(* Logix 5000 project; controller PBS_Perfusion vendor 1 type 14 code 217 rev 32.14; software revision 32.03; part 18 of 27 *)
(* tags used below, declared in another part *)
   Inp_OpenLS : BOOL;   // Valve Open Limit Switch 1=confirmed fully open
   Inp_ClosedLS : BOOL;   // Valve Closed Limit Switch 1=confirmed fully closed
   Inp_ActuatorFault : BOOL;   // Valve Actuator Fault (overload, etc.), 0=OK, 1=Fault)
   Inp_IntlkOK : BOOL;   // 1=Interlocks OK, Pulse Output Valve can be moved
   Inp_NBIntlkOK : BOOL;   // 1=Non-Bypassable Interlocks OK, Pulse Output Valve can be moved
   Inp_IntlkAvail : BOOL;   // 1 = Interlock Availibility OK
   Inp_IOFault : BOOL;   // Input / Output Communication Status 0=OK, 1=fail
   Inp_Sim : BOOL;   // 1=I/O are being simulated, set output CV to 0.0, ignore I/O Fault
   Inp_Reset : BOOL;   // 1=Reset shed latches and cleared alarms
   Cfg_ShedHold : BOOL;   // 1=Hold Output on Interlock or bad PV, 0=Go to Cfg_IntlkCV
   Cfg_ShedOnIOFault : BOOL;   // 1=Take shed action (hold or interlock CV) on I/O Fault
   Cfg_SkipRoCLim : BOOL;   // 1=Skip RoC Limiting in Intlk, Maint, Ovrd modes
   Cfg_SetTrack : BOOL;   // 1=PSets track OSets in Oper, OSets track PSets in Prog, 0=no tracking
   Cfg_SetTrackOvrdHand : BOOL;   // 1=Prog/Oper Settings track Override/Hand CV
   Cfg_HasOpenLS : BOOL;   // 1=Valve provides an Open Limit Switch signal
   Cfg_HasClosedLS : BOOL;   // 1=Valve provides a Closed Limit Switch signal
   Cfg_UseOpenLS : BOOL;   // 1=Valve Open LS should be used for open/closed status
   Cfg_UseClosedLS : BOOL;   // 1=Valve Closed LS should be used for open/closed status
   Cfg_LSFail : BOOL;   // 1=both switches ON=fail, 0=both switches OFF=fail
   Cfg_MinCV : REAL;   // Minimum CV (in CV EU, for limiting)
   Cfg_MaxCV : REAL;   // Maximum CV (in CV EU, for limiting)
   Cfg_CVRoCLimInc : REAL;   // CV Rate of Change Limit, Increasing, (EU/sec, 0=unlimited)
   Cfg_CVRoCLimDec : REAL;   // CV Rate of Change Limit, Decreasing, (EU/sec, 0=unlimited)
   Cfg_IntlkCV : REAL;   // CV (target in EU) when interlocked (if not Cfg_ShedHold)
   Cfg_CVEUMin : REAL;   // CV Minimum in Engineering Units (for scaling)
   Cfg_CVEUMax : REAL;   // CV Maximum in Engineering Units (for scaling)
   Cfg_CVRawMin : REAL;   // CV Minimum in I/O (raw) Units (for scaling)
   Cfg_CVRawMax : REAL;   // CV Maximum in I/O (raw) Units (for scaling)
   Cfg_CycleT : REAL;   // Open and Close Pulse Output overall period (s)
   Cfg_OpenRate : REAL;   // Rate at which valve moves when opening (CV EU/sec)
   Cfg_CloseRate : REAL;   // Rate at which valve moves when closing (CV EU/sec)
   Cfg_MaxOnT : REAL;   // Open and Close Pulse Output maximum ON time (s)
   Cfg_MinOnT : REAL;   // Open and Close Pulse Output minimum ON time (s)
   Cfg_BumpT : REAL;   // Time to bump valve open or closed (by Oper) when Fdbk Bad (sec)
   Cfg_Deadtime : REAL;   // Additional time on first pulse after stop or direction change
   Cfg_MaxClosedPos : REAL;   // Position above which valve is assumed open if limit switches not used
   PSet_CV : REAL;   // Program Setting of Controlled Variable (output) (CV EU)
   XSet_CV : REAL;   // External Setting of Controlled Variable (output) (CV EU)
   PCmd_Reset : BOOL;   // Program Command to reset shed latches and cleared alarms
   XCmd_Reset : BOOL;   // External Command to reset shed latches and cleared alarms
   Out_CV : REAL;   // CV Output in Raw (I/O Card) Units
   Out_Open : BOOL;   // Pulse Output to drive valve Open
   Out_Close : BOOL;   // Pulse Output to drive valve closed
   Val_Pos : REAL;   // Valve actual position from feedback (CV EU)
   Val_CVSet : REAL;   // Value of selected CV Setting (before rate limiting, CV EU)
   Val_CVOut : REAL;   // Value of CV output (after clamping and ramping) (CV EU)
   SrcQ_IO : DINT;   // Source and Quality of primary I/O (enumeration)
   SrcQ : DINT;   // Source and Quality of primary Val/Sts (enumeration)
   Val_Fdbk : DINT;   // Device Feedback 0=Moving, 1=Closed, 2=Opened, 3=Limit Switch Failure
   Val_Sts : DINT;   // 0=AtTarget, 1=RampClose, 2=RampOpen, 3=Clamp@Min, 4=Clamp@Max, 5=BumpClose, 6=BumpOpen
   Val_Fault : DINT;   // Device Fault Status 0=none, 32=I/OFault, 34=CfgErr
   Val_NotifyAll : DINT;   // Highest Alarm prio and ack status this object + channel (enum)
   Val_UnackAlmC : DINT;   // Count of Unacknowledged Alarms
   Sts_CVInfNaN : BOOL;   // 1=Selected CV is Infinite or Not A Number (1.$, 1.#NaN)
   Sts_PosInfNaN : BOOL;   // 1=Inp_PosFdbk is Infinite or Not A Number (1.$, 1.#NaN)
   Sts_BumpOpen : BOOL;   // 1=Bump Open Requested or Active
   Sts_BumpClose : BOOL;   // 1=Bump Close Requested or Active
   Sts_Ramping : BOOL;   // 1=CV is ramping to target
   Sts_Clamped : BOOL;   // 1=CV Set is clamped at CVMin or CVMax
   Sts_SkipRoCLim : BOOL;   // 1=Rate of Change Limiting was skipped this scan (Maint, Ovrd, Intlk, Hand)
   Sts_Active : BOOL;   // 1=CV is greater than Cfg_MaxClosedPos, show valve symbol as "opened"
   Sts_Available : BOOL;   // 1=Pulse Output Valve available for control by automation (Prog)
   Sts_BypActive : BOOL;   // 1=Bypassing Active (Bypassed or Maintenance)
   Sts_LSFail : BOOL;   // 1=Limit Switch Overlap Failure
   Sts_NotRdy : BOOL;   // 1=Device Not Ready, see detail bits for reason
   Nrdy_CfgErr : BOOL;   // 1=Device Not Ready: Configuration Error
   Nrdy_Intlk : BOOL;   // 1=Device Not Ready: Interlock Not OK
   Nrdy_IOFault : BOOL;   // 1=Device Not Ready: I/O Fault (Shed Requires Reset)
   Nrdy_OoS : BOOL;   // 1=Device Not Ready: Device is Out of Service
   Sts_AlmInh : BOOL;   // 1=One or more Alarms Shelved, Disabled or Suppressed
   Sts_Err : BOOL;   // 1=Error in Config: see detail bits for reason
   Err_EU : BOOL;   // 1=Error in Config: Scaled CV EU Min = Max
   Err_Raw : BOOL;   // 1=Error in Config: Raw Output Scaling Min = Max
   Err_Alarm : BOOL;   // 1=Error in Config: Alarm Min On Time, Shelf Time, Severity
   Sts_Hand : ALIAS FOR CmdSrc.Sts_Hand;
   Sts_OoS : ALIAS FOR CmdSrc.Sts_OoS;
   Sts_Maint : ALIAS FOR CmdSrc.Sts_Maint;
   Sts_Ovrd : ALIAS FOR CmdSrc.Sts_Ovrd;
   Sts_Prog : ALIAS FOR CmdSrc.Sts_Prog;
   Sts_Oper : ALIAS FOR CmdSrc.Sts_Oper;
   Sts_RdyReset : ALIAS FOR ORdy_Reset;   // 1=A latched alarm or shed condition is ready to be reset
   Sts_RdyAck : BOOL;   // 1=An alarm is ready to be acknowledged
   Sts_IntlkTrip : ALIAS FOR IntlkTrip.Inp;   // 1=Status: CV held or forced by interlock NOT OK (1-shot)
   Sts_ActuatorFault : ALIAS FOR ActuatorFault.Inp;   // 1=Actuator Fault detected (input)
   Sts_IOFault : ALIAS FOR IOFault.Inp;   // 1=I/O Fault Status (0=OK, 1=Bad)
   P_ValveC : BOOL;   // Unique Parameter Name for auto - discovery
   CmdSrc : P_CmdSrc;   // Control / Command Source Selection
   IOFault : P_Alarm;   // I/O Fault Alarm
   IntlkTrip : P_Alarm;   // Interlock Trip Alarm
   Wrk_Notify : DINT;   // Buffer for building Val_Notify
   Wrk_Bypass : BOOL;   // Internal Bypassable Interlocks are Bypassed flag
   Wrk_CV : REAL;   // Working copy of Speed Reference (for limiting)
   Wrk_CVSet : REAL;   // Final selected CV to feed to RoC Limiter
   Wrk_CVOut : REAL;   // Working value of CV after Rate Limiting
   Wrk_IntlkTripONS : BOOL;   // Interlock Tripped This Scan
   Wrk_ScanTime : REAL;   // Seconds since previous scan
   Wrk_StepInc : REAL;   // Amount to increase CV (to valve pulse logic) this scan for rate limiting
   Wrk_Sts : DINT;   // Buffer for building Val_Sts
   Wrk_Fault : DINT;   // Buffer for building Val_Fault
   Wrk_SrcQ : DINT;   // Register for building Source / Quality enumeration
   ActuatorFault : P_Alarm;   // Actuator Fault Alarm (based on Actuator Fault Input)
   Wrk_RealChkDINT : DINT;   // REAL tag bit pattern as a DINT to check for Inf / NaN
   Wrk_Close : BOOL;   // Internal Close output -- before Sim
   Wrk_Open : BOOL;   // Internal Open output -- before Sim
   Wrk_CycleT : TIMER;   // Overall Cycle Timer for pulsed outputs
   Wrk_OKtoOpen : BOOL;   // OK to pulse Out_Open
   Wrk_OKtoClose : BOOL;   // OK to pulse Out_Close
   Wrk_OpenTime : REAL;   // Time to pulse Out_Open
   Wrk_CycleT_ms : DINT;   // Cycle Time in milliseconds (preset)
   Wrk_OpenTimePrev : DINT;   // Wrk_OpenTime from previous cycle
   Wrk_CloseTime : REAL;   // Time to pulse Out_Close
   Wrk_CloseTimePrev : REAL;   // Wrk_CloseTime from previous cycle
   Wrk_OpenFdbk : BOOL;   // 1=LS Feedback shows valve confirmed open
   Wrk_ClosedFdbk : BOOL;   // 1=LS Feedback shows valve confirmed closed
   Wrk_StepDec : REAL;   // Amount to decrease CV (to valve pulse logic) this scan for rate limiting
   Wrk_BumpClose : BOOL;   // Operator Bump Close requested
   Wrk_BumpOpen : BOOL;   // Operator Bump Open requested
   Wrk_BumpingOpen : BOOL;   // Operator Bump Open actively pulsing Out_Open
   Wrk_BumpingClose : BOOL;   // Operator Bump Close actively pulsing Out_Close
   Wrk_CycleActive : BOOL;   // Outputs are cycling; wait for cycle to complete
   Wrk_ShedIntlkCV : BOOL;   // Output CV being held at Interlock value
   Wrk_ShedHold : BOOL;   // Output CV being held at last good value
   OSet_CV : REAL;   // Operator Setting of Controlled Variable (output) (CV EU)
   OCmd_ResetAckAll : BOOL;   // Oper Cmd to reset shed latches and cleared alarms and acknowledge all alarms
   OCmd_Reset : BOOL;   // Oper Cmd to reset shed latches and cleared alarms
   OCmd_BumpClose : BOOL;   // Operator Command to bump valve closed (avail. if Fdbk Bad)
   OCmd_BumpOpen : BOOL;   // Operator Command to bump valve open (avail. if Fdbk Bad)
   ORdy_CV : BOOL;   // 1=Ready for OSet_CV (enables data entry field)
   ORdy_ResetAckAll : BOOL;   // 1=Ready for OCmd_ResetAckAll (enables HMI button)
   ORdy_Reset : BOOL;   // 1=Ready for OCmd_Reset (enables HMI button)
   MRdy_Check : BOOL;   // 1=Ready for MCmd_Check (enables HMI button)
   MRdy_Bypass : BOOL;   // 1=Ready for MCmd_Bypass (enables HMI button)
   ORdy_BumpClose : BOOL;   // 1=Ready for OCmd_BumpClose (enables HMI button)
   ORdy_BumpOpen : BOOL;   // 1=Ready for OCmd_BumpOpen (enables HMI button)
   Wrk_UnackAlmC : DINT;   // Buffer for building Val_UnackAlmC
   Val_Notify : DINT;   // Current Alarm Level and Acknowledgement (enumeration)
   ONS : DINT[3];
   REAL : DINT;
(* P_ValveC, continued *)

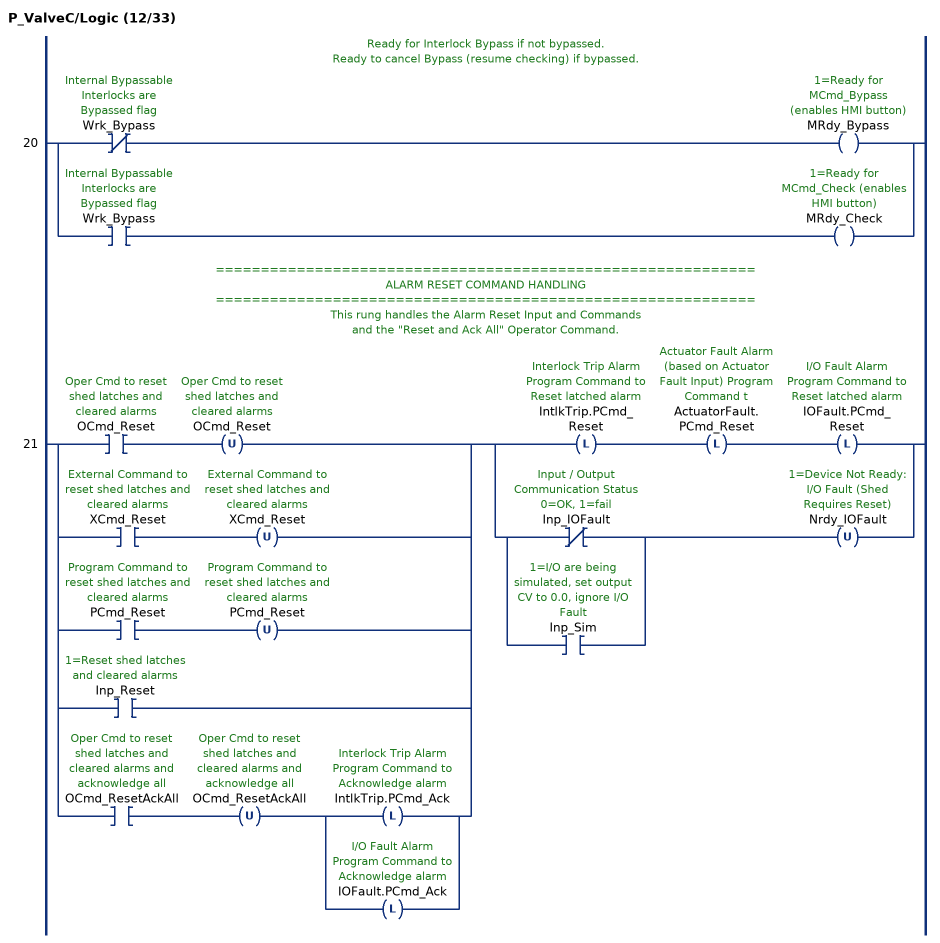
   [picture p394: P_ValveC/Logic rungs 20-21]
   // Ready for Interlock Bypass if not bypassed.
   // Ready to cancel Bypass (resume checking) if bypassed.
   20: [XIO(Wrk_Bypass) OTE(MRdy_Bypass) ,XIC(Wrk_Bypass) OTE(MRdy_Check) ];
   // ============================================================
   // ALARM RESET COMMAND HANDLING
   // ============================================================
   // This rung handles the Alarm Reset Input and Commands
   // and the "Reset and Ack All" Operator Command.
   21: [XIC(OCmd_Reset) OTU(OCmd_Reset) ,XIC(XCmd_Reset) OTU(XCmd_Reset) ,XIC(PCmd_Reset) OTU(PCmd_Reset) ,XIC(Inp_Reset) ,XIC(OCmd_ResetAckAll) OTU(OCmd_ResetAckAll) [OTL(IntlkTrip.PCmd_Ack) ,OTL(IOFault.PCmd_Ack) ] ][OTL(IntlkTrip.PCmd_Reset) OTL(ActuatorFault.PCmd_Reset) OTL(IOFault.PCmd_Reset) ,[XIO(Inp_IOFault) ,XIC(Inp_Sim) ] OTU(Nrdy_IOFault) ];
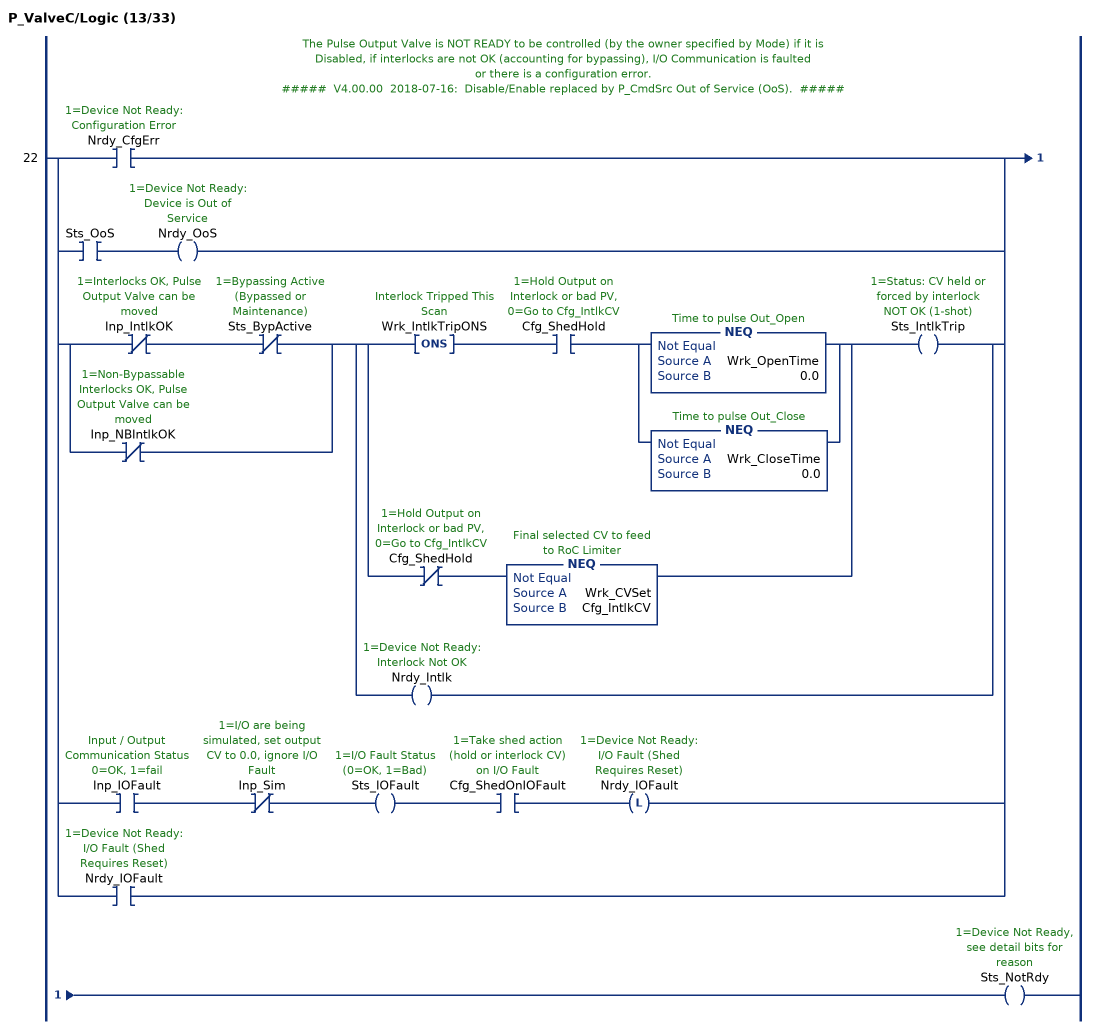
   // The Pulse Output Valve is NOT READY to be controlled (by the owner specified by Mode) if it is
   // Disabled, if interlocks are not OK (accounting for bypassing), I/O Communication is faulted
   // or there is a configuration error.
   // #####  V4.00.00  2018-07-16:  Disable/Enable replaced by P_CmdSrc Out of Service (OoS).  #####
   22: [XIC(Nrdy_CfgErr) ,XIC(Sts_OoS) OTE(Nrdy_OoS) ,[XIO(Inp_IntlkOK) XIO(Sts_BypActive) ,XIO(Inp_NBIntlkOK) ] [[ONS(Wrk_IntlkTripONS) XIC(Cfg_ShedHold) [NEQ(Wrk_OpenTime,0.0) ,NEQ(Wrk_CloseTime,0.0) ] ,XIO(Cfg_ShedHold) NEQ(Wrk_CVSet,Cfg_IntlkCV) ] OTE(Sts_IntlkTrip) ,OTE(Nrdy_Intlk) ] ,XIC(Inp_IOFault) XIO(Inp_Sim) OTE(Sts_IOFault) XIC(Cfg_ShedOnIOFault) OTL(Nrdy_IOFault) ,XIC(Nrdy_IOFault) ]OTE(Sts_NotRdy);
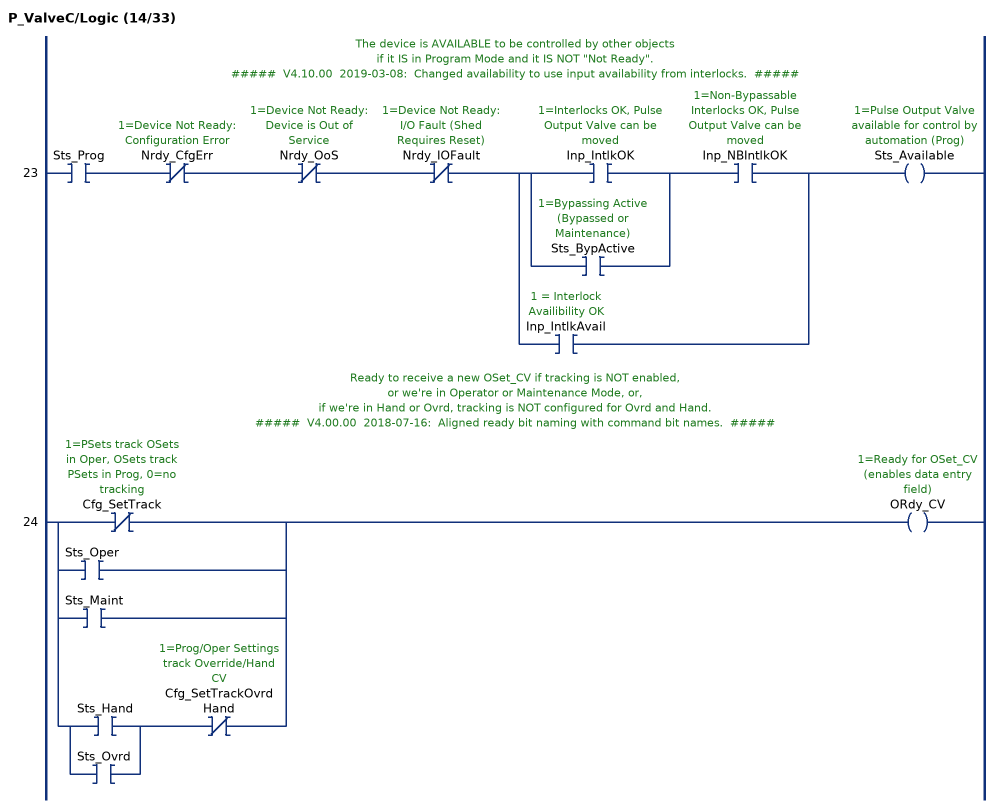
   // The device is AVAILABLE to be controlled by other objects
   // if it IS in Program Mode and it IS NOT "Not Ready".
   // #####  V4.10.00  2019-03-08:  Changed availability to use input availability from interlocks.  #####
   23: XIC(Sts_Prog)XIO(Nrdy_CfgErr)XIO(Nrdy_OoS)XIO(Nrdy_IOFault)[[XIC(Inp_IntlkOK) ,XIC(Sts_BypActive) ] XIC(Inp_NBIntlkOK) ,XIC(Inp_IntlkAvail) ]OTE(Sts_Available);
   // Ready to receive a new OSet_CV if tracking is NOT enabled,
   // or we're in Operator or Maintenance Mode, or,
   // if we're in Hand or Ovrd, tracking is NOT configured for Ovrd and Hand.
   // #####  V4.00.00  2018-07-16:  Aligned ready bit naming with command bit names.  #####
   24: [XIO(Cfg_SetTrack) ,XIC(Sts_Oper) ,XIC(Sts_Maint) ,[XIC(Sts_Hand) ,XIC(Sts_Ovrd) ] XIO(Cfg_SetTrackOvrdHand) ]OTE(ORdy_CV);
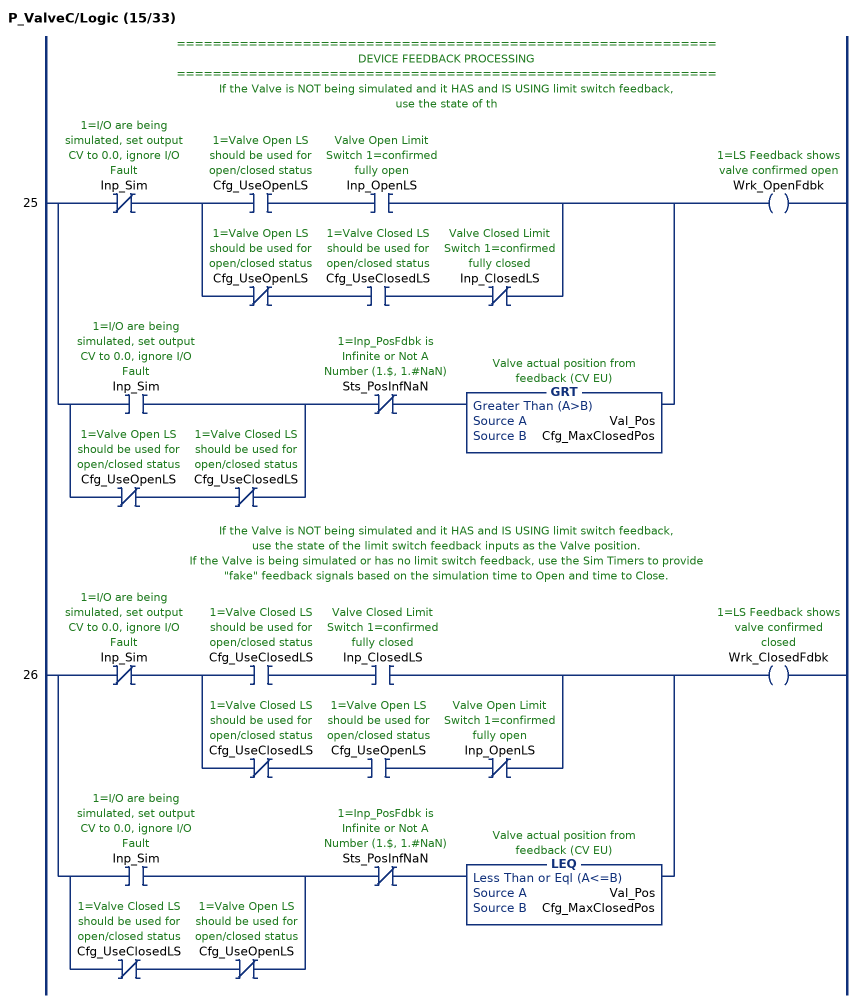
   // ============================================================
   // DEVICE FEEDBACK PROCESSING
   // ============================================================
   // If the Valve is NOT being simulated and it HAS and IS USING limit switch feedback,
   // use the state of th
   25: [XIO(Inp_Sim) [XIC(Cfg_UseOpenLS) XIC(Inp_OpenLS) ,XIO(Cfg_UseOpenLS) XIC(Cfg_UseClosedLS) XIO(Inp_ClosedLS) ] ,[XIC(Inp_Sim) ,XIO(Cfg_UseOpenLS) XIO(Cfg_UseClosedLS) ] XIO(Sts_PosInfNaN) GRT(Val_Pos,Cfg_MaxClosedPos) ]OTE(Wrk_OpenFdbk);
   // If the Valve is NOT being simulated and it HAS and IS USING limit switch feedback,
   // use the state of the limit switch feedback inputs as the Valve position.
   // If the Valve is being simulated or has no limit switch feedback, use the Sim Timers to provide
   // "fake" feedback signals based on the simulation time to Open and time to Close.
   26: [XIO(Inp_Sim) [XIC(Cfg_UseClosedLS) XIC(Inp_ClosedLS) ,XIO(Cfg_UseClosedLS) XIC(Cfg_UseOpenLS) XIO(Inp_OpenLS) ] ,[XIC(Inp_Sim) ,XIO(Cfg_UseClosedLS) XIO(Cfg_UseOpenLS) ] XIO(Sts_PosInfNaN) LEQ(Val_Pos,Cfg_MaxClosedPos) ]OTE(Wrk_ClosedFdbk);
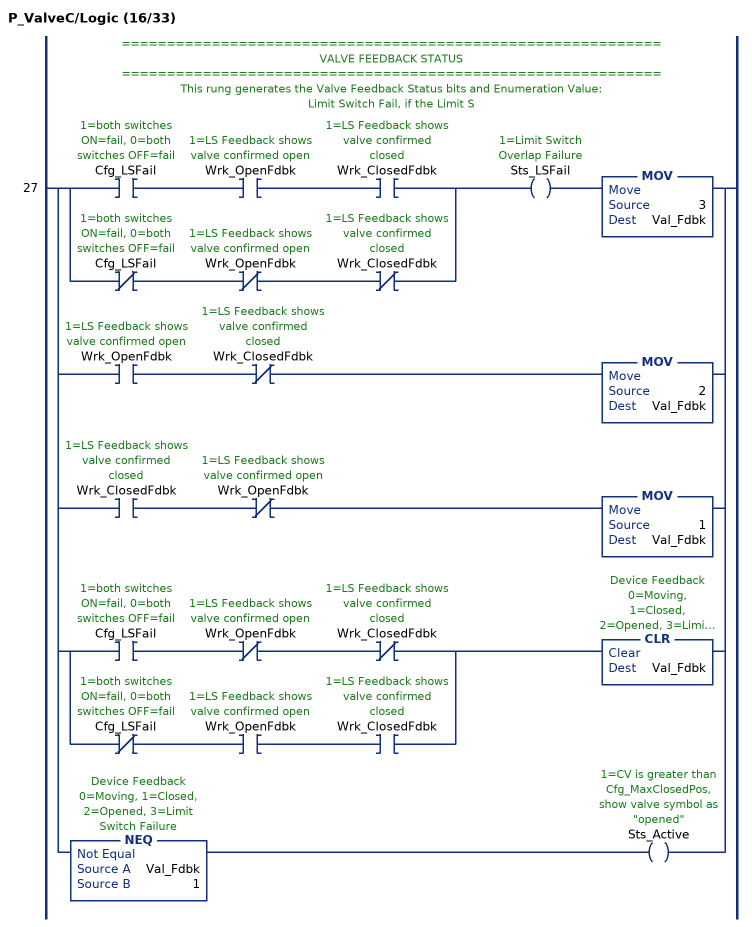
   // ============================================================
   // VALVE FEEDBACK STATUS
   // ============================================================
   // This rung generates the Valve Feedback Status bits and Enumeration Value:
   // Limit Switch Fail, if the Limit S
   27: [[XIC(Cfg_LSFail) XIC(Wrk_OpenFdbk) XIC(Wrk_ClosedFdbk) ,XIO(Cfg_LSFail) XIO(Wrk_OpenFdbk) XIO(Wrk_ClosedFdbk) ] OTE(Sts_LSFail) MOV(3,Val_Fdbk) ,XIC(Wrk_OpenFdbk) XIO(Wrk_ClosedFdbk) MOV(2,Val_Fdbk) ,XIC(Wrk_ClosedFdbk) XIO(Wrk_OpenFdbk) MOV(1,Val_Fdbk) ,[XIC(Cfg_LSFail) XIO(Wrk_OpenFdbk) XIO(Wrk_ClosedFdbk) ,XIO(Cfg_LSFail) XIC(Wrk_OpenFdbk) XIC(Wrk_ClosedFdbk) ] CLR(Val_Fdbk) ,NEQ(Val_Fdbk,1) OTE(Sts_Active) ];
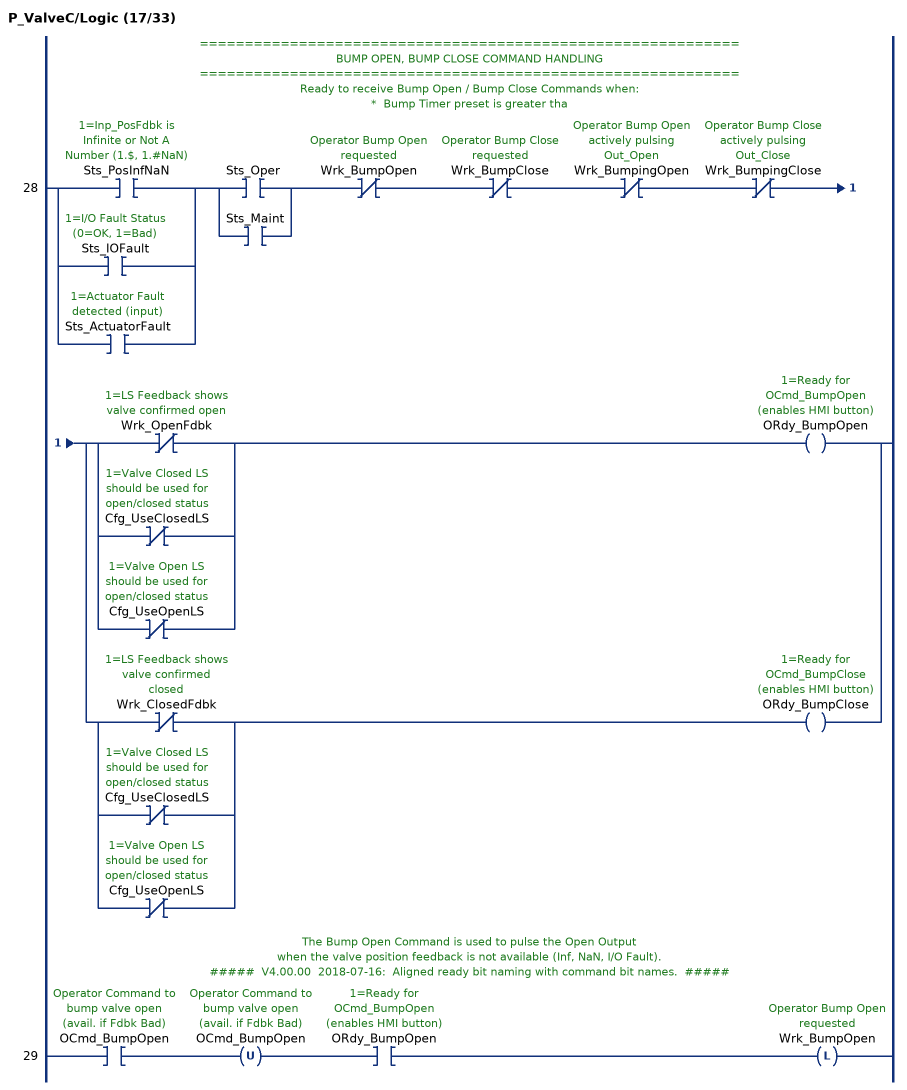
   // ============================================================
   // BUMP OPEN, BUMP CLOSE COMMAND HANDLING
   // ============================================================
   // Ready to receive Bump Open / Bump Close Commands when:
   // *  Bump Timer preset is greater tha
   28: [XIC(Sts_PosInfNaN) ,XIC(Sts_IOFault) ,XIC(Sts_ActuatorFault) ][XIC(Sts_Oper) ,XIC(Sts_Maint) ]XIO(Wrk_BumpOpen)XIO(Wrk_BumpClose)XIO(Wrk_BumpingOpen)XIO(Wrk_BumpingClose)[[XIO(Wrk_OpenFdbk) ,XIO(Cfg_UseClosedLS) ,XIO(Cfg_UseOpenLS) ] OTE(ORdy_BumpOpen) ,[XIO(Wrk_ClosedFdbk) ,XIO(Cfg_UseClosedLS) ,XIO(Cfg_UseOpenLS) ] OTE(ORdy_BumpClose) ];
   // The Bump Open Command is used to pulse the Open Output
   // when the valve position feedback is not available (Inf, NaN, I/O Fault).
   // #####  V4.00.00  2018-07-16:  Aligned ready bit naming with command bit names.  #####
   29: XIC(OCmd_BumpOpen)OTU(OCmd_BumpOpen)XIC(ORdy_BumpOpen)OTL(Wrk_BumpOpen);
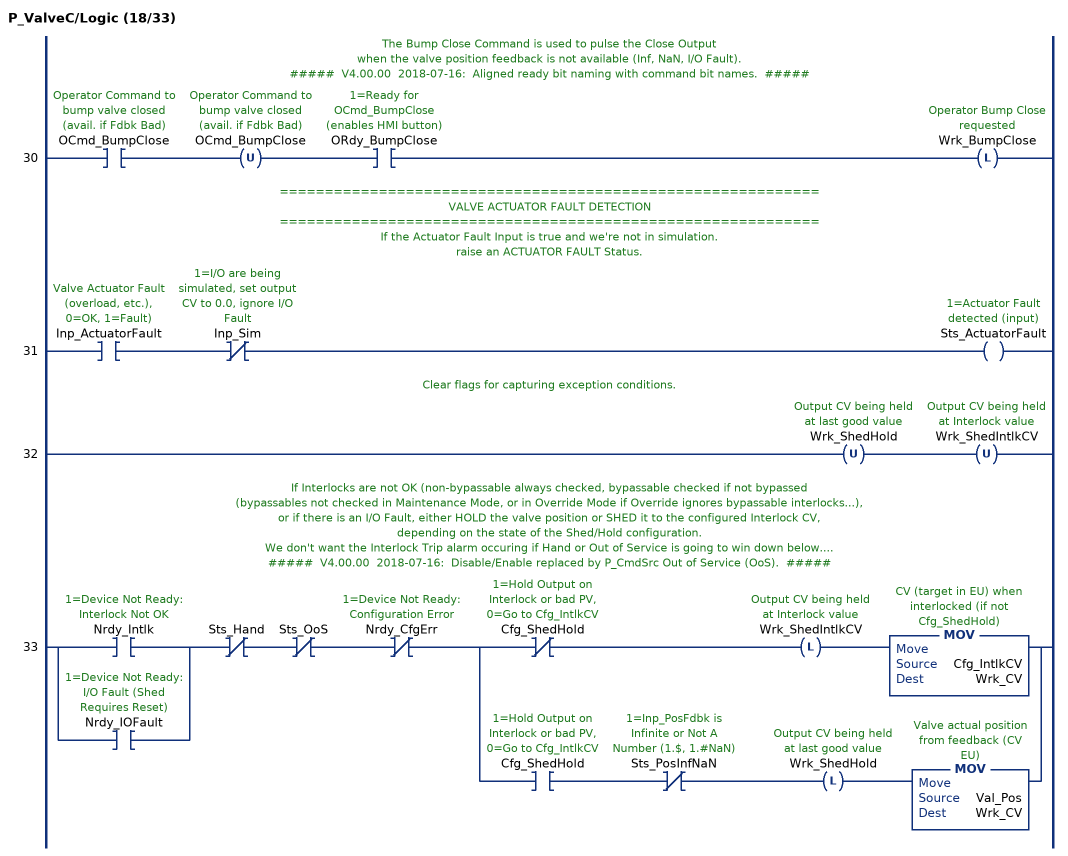
   // The Bump Close Command is used to pulse the Close Output
   // when the valve position feedback is not available (Inf, NaN, I/O Fault).
   // #####  V4.00.00  2018-07-16:  Aligned ready bit naming with command bit names.  #####
   30: XIC(OCmd_BumpClose)OTU(OCmd_BumpClose)XIC(ORdy_BumpClose)OTL(Wrk_BumpClose);
   // ============================================================
   // VALVE ACTUATOR FAULT DETECTION
   // ============================================================
   // If the Actuator Fault Input is true and we're not in simulation.
   // raise an ACTUATOR FAULT Status.
   31: XIC(Inp_ActuatorFault)XIO(Inp_Sim)OTE(Sts_ActuatorFault);
   // Clear flags for capturing exception conditions.
   32: OTU(Wrk_ShedHold)OTU(Wrk_ShedIntlkCV);
   // If Interlocks are not OK (non-bypassable always checked, bypassable checked if not bypassed
   // (bypassables not checked in Maintenance Mode, or in Override Mode if Override ignores bypassable interlocks...),
   // or if there is an I/O Fault, either HOLD the valve position or SHED it to the configured Interlock CV,
   // depending on the state of the Shed/Hold configuration.
   // We don't want the Interlock Trip alarm occuring if Hand or Out of Service is going to win down below....
   // #####  V4.00.00  2018-07-16:  Disable/Enable replaced by P_CmdSrc Out of Service (OoS).  #####
   33: [XIC(Nrdy_Intlk) ,XIC(Nrdy_IOFault) ]XIO(Sts_Hand)XIO(Sts_OoS)XIO(Nrdy_CfgErr)[XIO(Cfg_ShedHold) OTL(Wrk_ShedIntlkCV) MOV(Cfg_IntlkCV,Wrk_CV) ,XIC(Cfg_ShedHold) XIO(Sts_PosInfNaN) OTL(Wrk_ShedHold) MOV(Val_Pos,Wrk_CV) ];
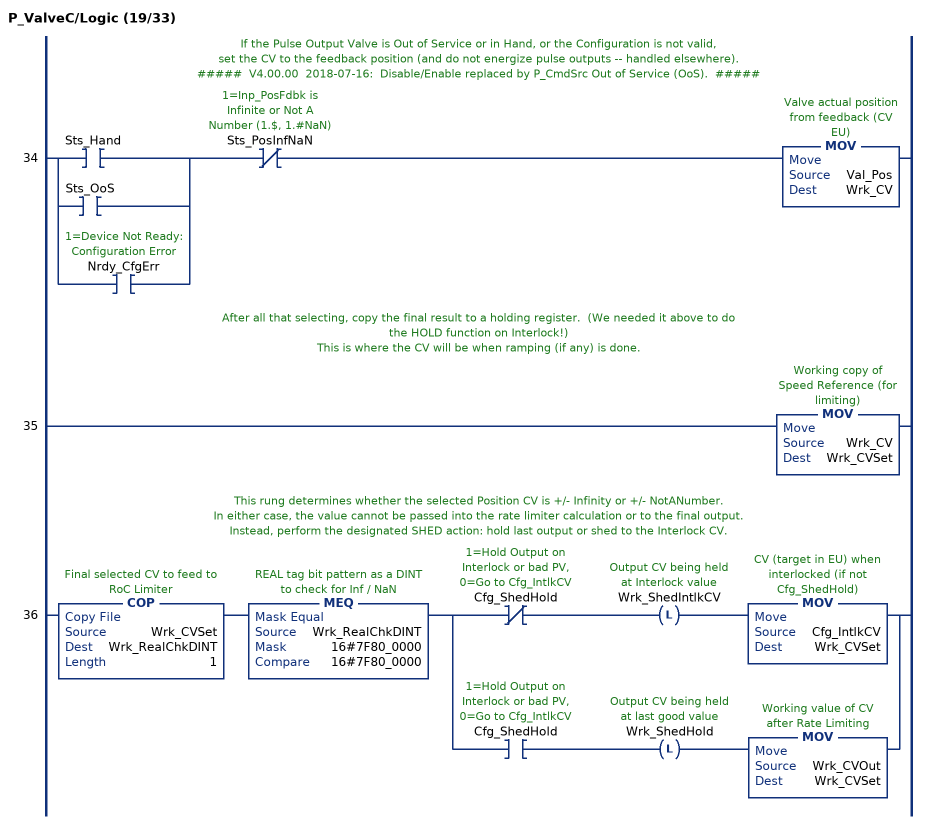
   // If the Pulse Output Valve is Out of Service or in Hand, or the Configuration is not valid,
   // set the CV to the feedback position (and do not energize pulse outputs -- handled elsewhere).
   // #####  V4.00.00  2018-07-16:  Disable/Enable replaced by P_CmdSrc Out of Service (OoS).  #####
   34: [XIC(Sts_Hand) ,XIC(Sts_OoS) ,XIC(Nrdy_CfgErr) ]XIO(Sts_PosInfNaN)MOV(Val_Pos,Wrk_CV);
   // After all that selecting, copy the final result to a holding register.  (We needed it above to do
   // the HOLD function on Interlock!)
   // This is where the CV will be when ramping (if any) is done.
   35: MOV(Wrk_CV,Wrk_CVSet);
   // This rung determines whether the selected Position CV is +/- Infinity or +/- NotANumber.
   // In either case, the value cannot be passed into the rate limiter calculation or to the final output.
   // Instead, perform the designated SHED action: hold last output or shed to the Interlock CV.
   36: COP(Wrk_CVSet,Wrk_RealChkDINT,1)MEQ(Wrk_RealChkDINT,16#7F80_0000,16#7F80_0000)[XIO(Cfg_ShedHold) OTL(Wrk_ShedIntlkCV) MOV(Cfg_IntlkCV,Wrk_CVSet) ,XIC(Cfg_ShedHold) OTL(Wrk_ShedHold) MOV(Wrk_CVOut,Wrk_CVSet) ];
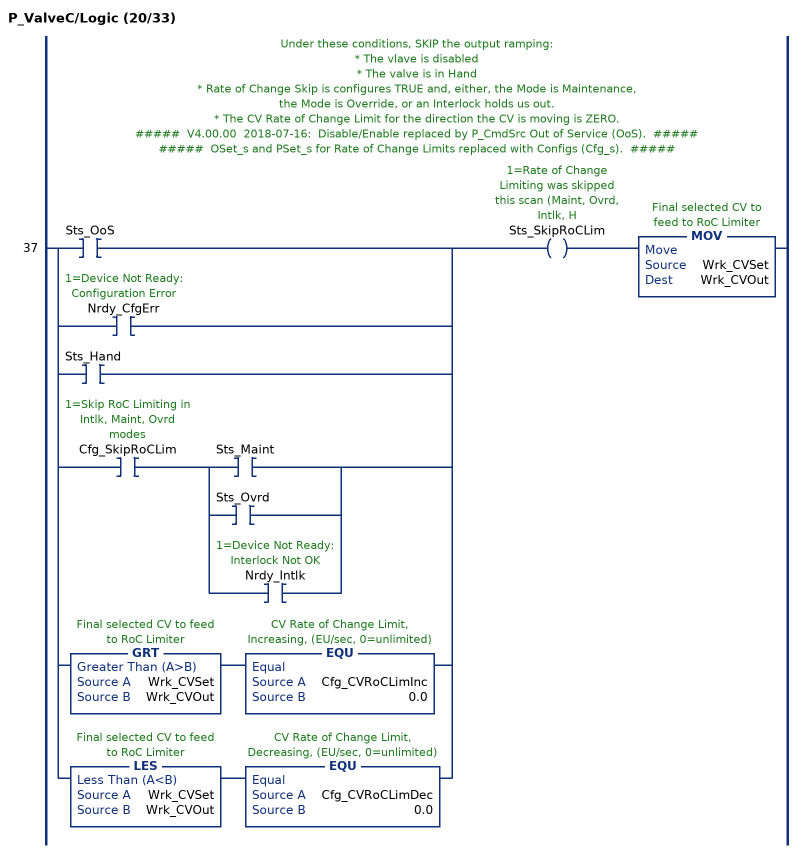
   // Under these conditions, SKIP the output ramping:
   // * The vlave is disabled
   // * The valve is in Hand
   // * Rate of Change Skip is configures TRUE and, either, the Mode is Maintenance,
   // the Mode is Override, or an Interlock holds us out.
   // * The CV Rate of Change Limit for the direction the CV is moving is ZERO.
   // #####  V4.00.00  2018-07-16:  Disable/Enable replaced by P_CmdSrc Out of Service (OoS).  #####
   // #####  OSet_s and PSet_s for Rate of Change Limits replaced with Configs (Cfg_s).  #####
   37: [XIC(Sts_OoS) ,XIC(Nrdy_CfgErr) ,XIC(Sts_Hand) ,XIC(Cfg_SkipRoCLim) [XIC(Sts_Maint) ,XIC(Sts_Ovrd) ,XIC(Nrdy_Intlk) ] ,GRT(Wrk_CVSet,Wrk_CVOut) EQU(Cfg_CVRoCLimInc,0.0) ,LES(Wrk_CVSet,Wrk_CVOut) EQU(Cfg_CVRoCLimDec,0.0) ]OTE(Sts_SkipRoCLim)MOV(Wrk_CVSet,Wrk_CVOut);
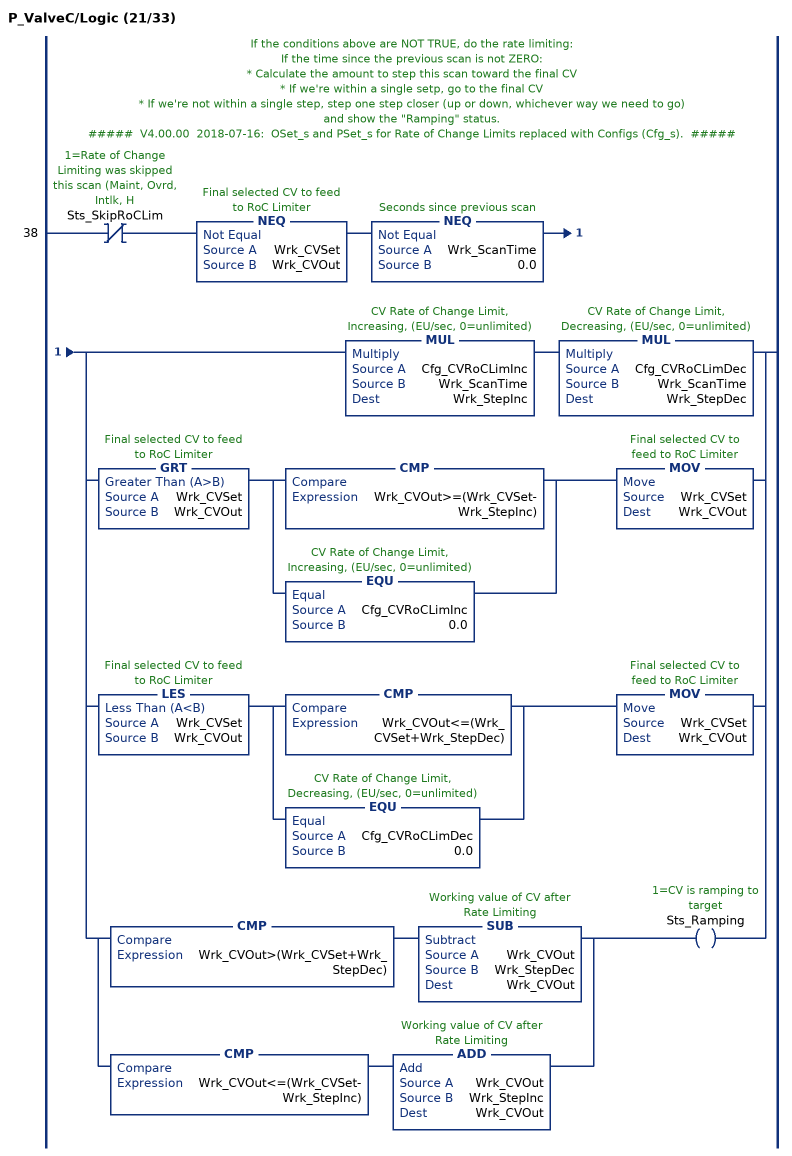
   // If the conditions above are NOT TRUE, do the rate limiting:
   // If the time since the previous scan is not ZERO:
   // * Calculate the amount to step this scan toward the final CV
   // * If we're within a single setp, go to the final CV
   // * If we're not within a single step, step one step closer (up or down, whichever way we need to go)
   // and show the "Ramping" status.
   // #####  V4.00.00  2018-07-16:  OSet_s and PSet_s for Rate of Change Limits replaced with Configs (Cfg_s).  #####
   38: XIO(Sts_SkipRoCLim)NEQ(Wrk_CVSet,Wrk_CVOut)NEQ(Wrk_ScanTime,0.0)[MUL(Cfg_CVRoCLimInc,Wrk_ScanTime,Wrk_StepInc) MUL(Cfg_CVRoCLimDec,Wrk_ScanTime,Wrk_StepDec) ,GRT(Wrk_CVSet,Wrk_CVOut) [CMP(Wrk_CVOut>=(Wrk_CVSet-Wrk_StepInc)) ,EQU(Cfg_CVRoCLimInc,0.0) ] MOV(Wrk_CVSet,Wrk_CVOut) ,LES(Wrk_CVSet,Wrk_CVOut) [CMP(Wrk_CVOut<=(Wrk_CVSet+Wrk_StepDec)) ,EQU(Cfg_CVRoCLimDec,0.0) ] MOV(Wrk_CVSet,Wrk_CVOut) ,[CMP(Wrk_CVOut>(Wrk_CVSet+Wrk_StepDec)) SUB(Wrk_CVOut,Wrk_StepDec,Wrk_CVOut) ,CMP(Wrk_CVOut<=(Wrk_CVSet-Wrk_StepInc)) ADD(Wrk_CVOut,Wrk_StepInc,Wrk_CVOut) ] OTE(Sts_Ramping) ];
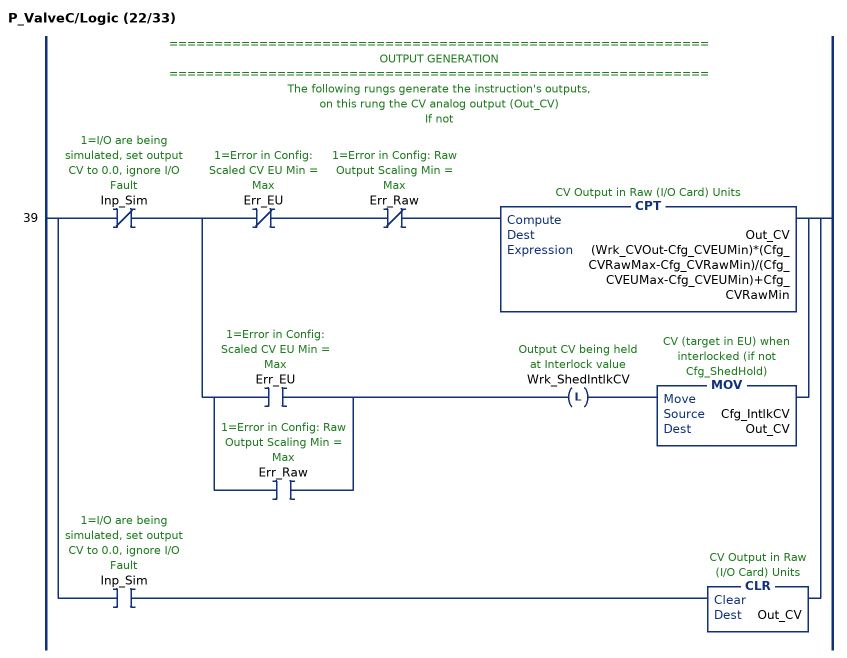
   // ============================================================
   // OUTPUT GENERATION
   // ============================================================
   // The following rungs generate the instruction's outputs,
   // on this rung the CV analog output (Out_CV)
   // If not
   39: [XIO(Inp_Sim) [XIO(Err_EU) XIO(Err_Raw) CPT(Out_CV,(Wrk_CVOut-Cfg_CVEUMin)*(Cfg_CVRawMax-Cfg_CVRawMin)/(Cfg_CVEUMax-Cfg_CVEUMin)+Cfg_CVRawMin) ,[XIC(Err_EU) ,XIC(Err_Raw) ] OTL(Wrk_ShedIntlkCV) MOV(Cfg_IntlkCV,Out_CV) ] ,XIC(Inp_Sim) CLR(Out_CV) ];
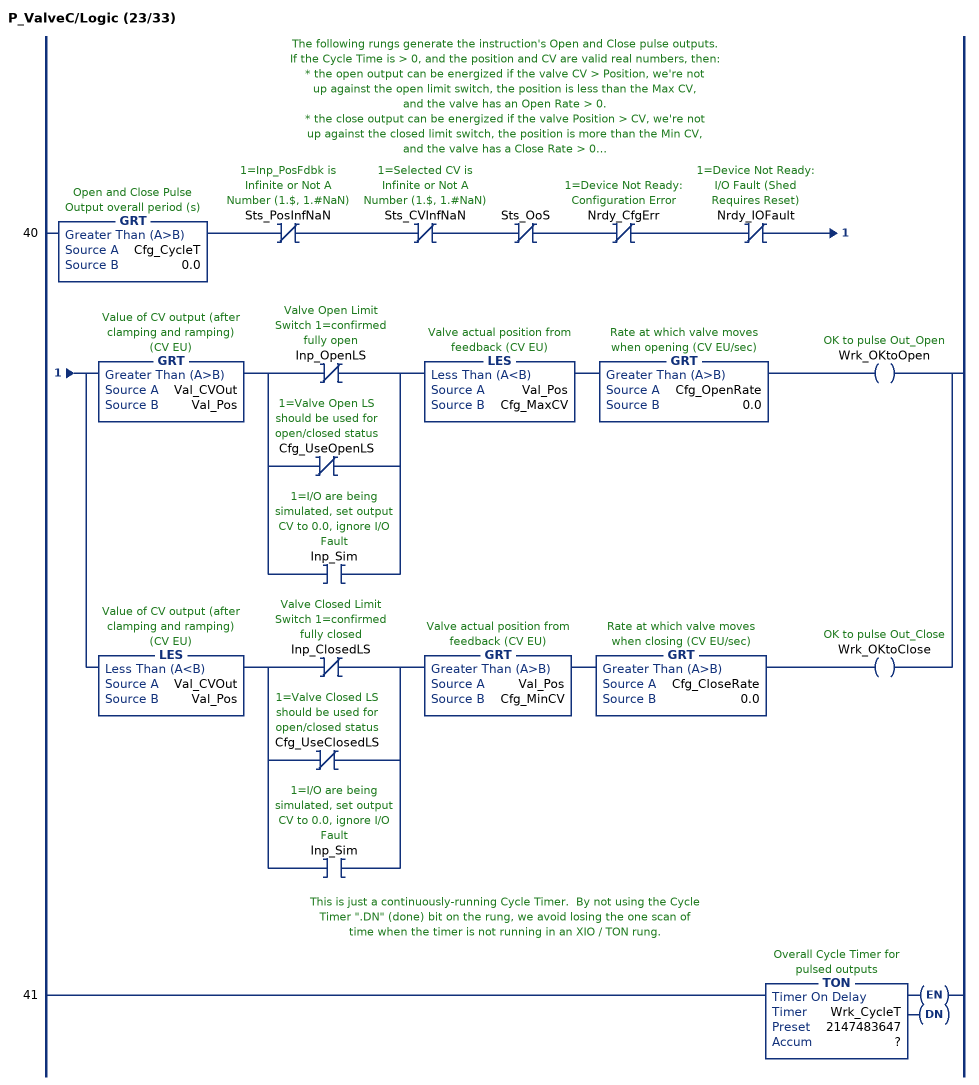
   // The following rungs generate the instruction's Open and Close pulse outputs.
   // If the Cycle Time is > 0, and the position and CV are valid real numbers, then:
   // * the open output can be energized if the valve CV > Position, we're not
   // up against the open limit switch, the position is less than the Max CV,
   // and the valve has an Open Rate > 0.
   // * the close output can be energized if the valve Position > CV, we're not
   // up against the closed limit switch, the position is more than the Min CV,
   // and the valve has a Close Rate > 0.
   // #####  V4.00.00  2018-07-16:  Disable/Enable replaced by P_CmdSrc Out of Service (OoS).  #####
   40: GRT(Cfg_CycleT,0.0)XIO(Sts_PosInfNaN)XIO(Sts_CVInfNaN)XIO(Sts_OoS)XIO(Nrdy_CfgErr)XIO(Nrdy_IOFault)[GRT(Val_CVOut,Val_Pos) [XIO(Inp_OpenLS) ,XIO(Cfg_UseOpenLS) ,XIC(Inp_Sim) ] LES(Val_Pos,Cfg_MaxCV) GRT(Cfg_OpenRate,0.0) OTE(Wrk_OKtoOpen) ,LES(Val_CVOut,Val_Pos) [XIO(Inp_ClosedLS) ,XIO(Cfg_UseClosedLS) ,XIC(Inp_Sim) ] GRT(Val_Pos,Cfg_MinCV) GRT(Cfg_CloseRate,0.0) OTE(Wrk_OKtoClose) ];
   // This is just a continuously-running Cycle Timer.  By not using the Cycle
   // Timer ".DN" (done) bit on the rung, we avoid losing the one scan of
   // time when the timer is not running in an XIO / TON rung.
   41: TON(Wrk_CycleT,?,?);
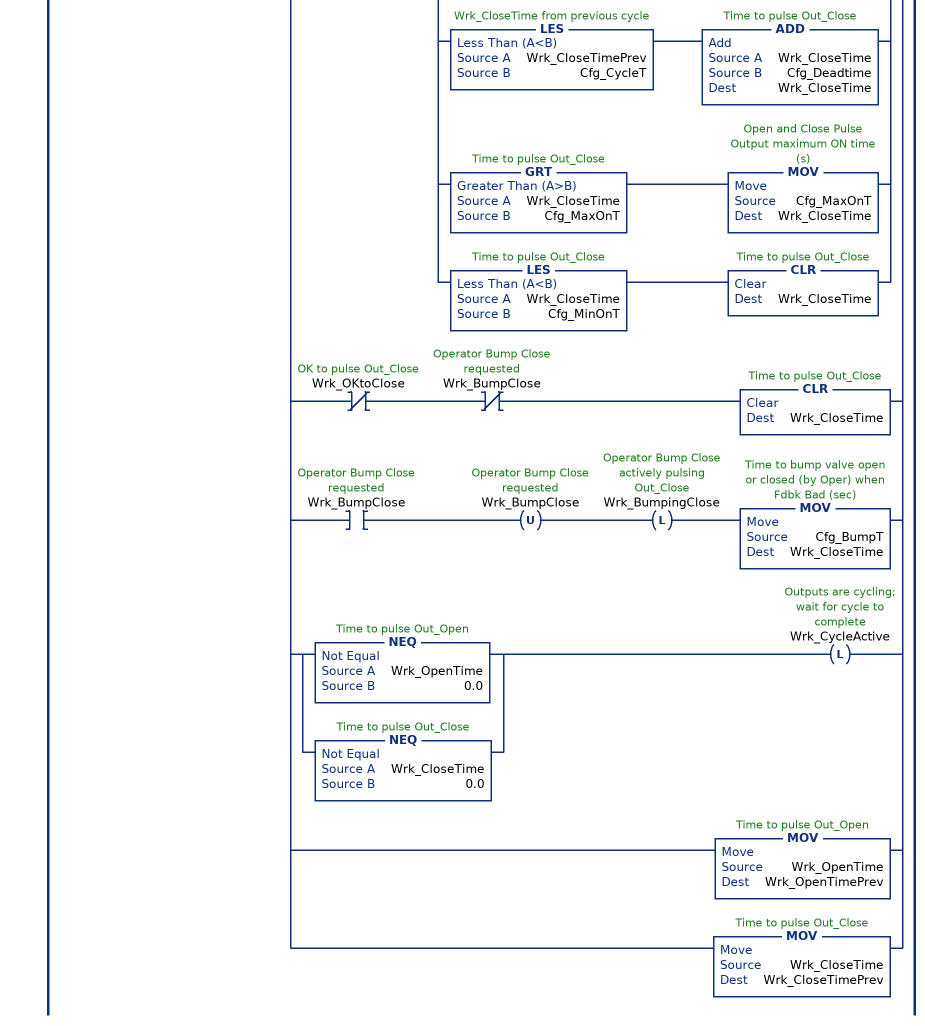
   // When the Cycle completes, calculate a new Open Time (time to pulse the
   // Open output) and Close Time (time to pulse the Close output).
   // Details of this calculation are in the Instruction Help for the POSP built-in
   // instruction, from which this logic is derived.
   42: [GEQ(Wrk_CycleT.ACC,Wrk_CycleT_ms) ,XIO(Wrk_CycleActive) ][OTU(Wrk_CycleActive) OTU(Wrk_BumpingOpen) OTU(Wrk_BumpingClose) CLR(Wrk_CycleT.ACC) ,XIC(Wrk_OKtoOpen) [CPT(Wrk_OpenTime,(Val_CVOut-Val_Pos)/Cfg_OpenRate) ,LES(Wrk_OpenTimePrev,Cfg_CycleT) ADD(Wrk_OpenTime,Cfg_Deadtime,Wrk_OpenTime) ,GRT(Wrk_OpenTime,Cfg_MaxOnT) MOV(Cfg_MaxOnT,Wrk_OpenTime) ,LES(Wrk_OpenTime,Cfg_MinOnT) CLR(Wrk_OpenTime) ] ,XIO(Wrk_OKtoOpen) XIO(Wrk_BumpOpen) CLR(Wrk_OpenTime) ,XIC(Wrk_BumpOpen) OTU(Wrk_BumpOpen) OTL(Wrk_BumpingOpen) MOV(Cfg_BumpT,Wrk_OpenTime) ,XIC(Wrk_OKtoClose) [CPT(Wrk_CloseTime,(Val_Pos-Val_CVOut)/Cfg_CloseRate) ,LES(Wrk_CloseTimePrev,Cfg_CycleT) ADD(Wrk_CloseTime,Cfg_Deadtime,Wrk_CloseTime) ,GRT(Wrk_CloseTime,Cfg_MaxOnT) MOV(Cfg_MaxOnT,Wrk_CloseTime) ,LES(Wrk_CloseTime,Cfg_MinOnT) CLR(Wrk_CloseTime) ] ,XIO(Wrk_OKtoClose) XIO(Wrk_BumpClose) CLR(Wrk_CloseTime) ,XIC(Wrk_BumpClose) OTU(Wrk_BumpClose) OTL(Wrk_BumpingClose) MOV(Cfg_BumpT,Wrk_CloseTime) ,[NEQ(Wrk_OpenTime,0.0) ,NEQ(Wrk_CloseTime,0.0) ] OTL(Wrk_CycleActive) ,MOV(Wrk_OpenTime,Wrk_OpenTimePrev) ,MOV(Wrk_CloseTime,Wrk_CloseTimePrev) ];
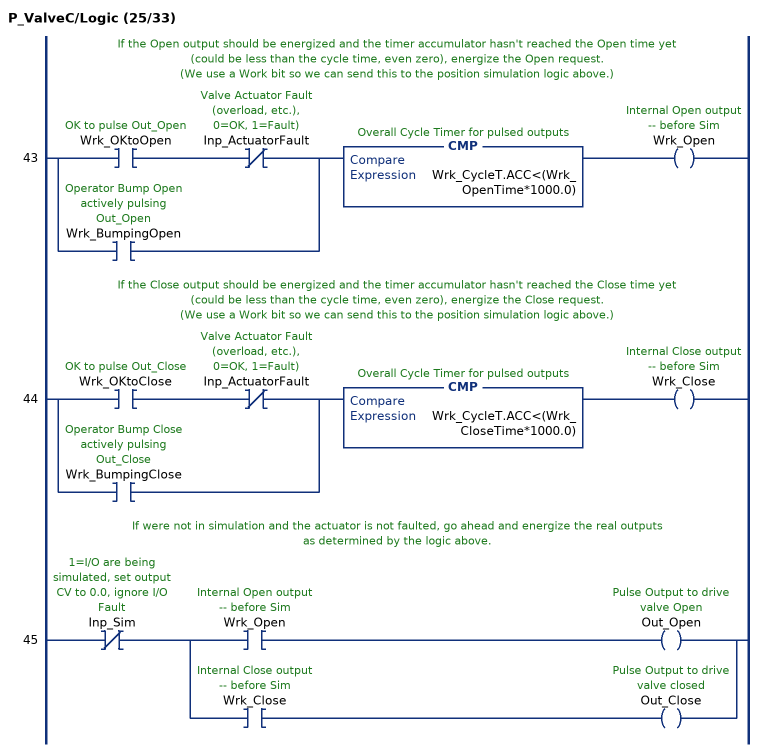
   // If the Open output should be energized and the timer accumulator hasn't reached the Open time yet
   // (could be less than the cycle time, even zero), energize the Open request.
   // (We use a Work bit so we can send this to the position simulation logic above.)
   43: [XIC(Wrk_OKtoOpen) XIO(Inp_ActuatorFault) ,XIC(Wrk_BumpingOpen) ]CMP(Wrk_CycleT.ACC<(Wrk_OpenTime*1000.0))OTE(Wrk_Open);
   // If the Close output should be energized and the timer accumulator hasn't reached the Close time yet
   // (could be less than the cycle time, even zero), energize the Close request.
   // (We use a Work bit so we can send this to the position simulation logic above.)
   44: [XIC(Wrk_OKtoClose) XIO(Inp_ActuatorFault) ,XIC(Wrk_BumpingClose) ]CMP(Wrk_CycleT.ACC<(Wrk_CloseTime*1000.0))OTE(Wrk_Close);
   // If were not in simulation and the actuator is not faulted, go ahead and energize the real outputs
   // as determined by the logic above.
   45: XIO(Inp_Sim)[XIC(Wrk_Open) OTE(Out_Open) ,XIC(Wrk_Close) OTE(Out_Close) ];
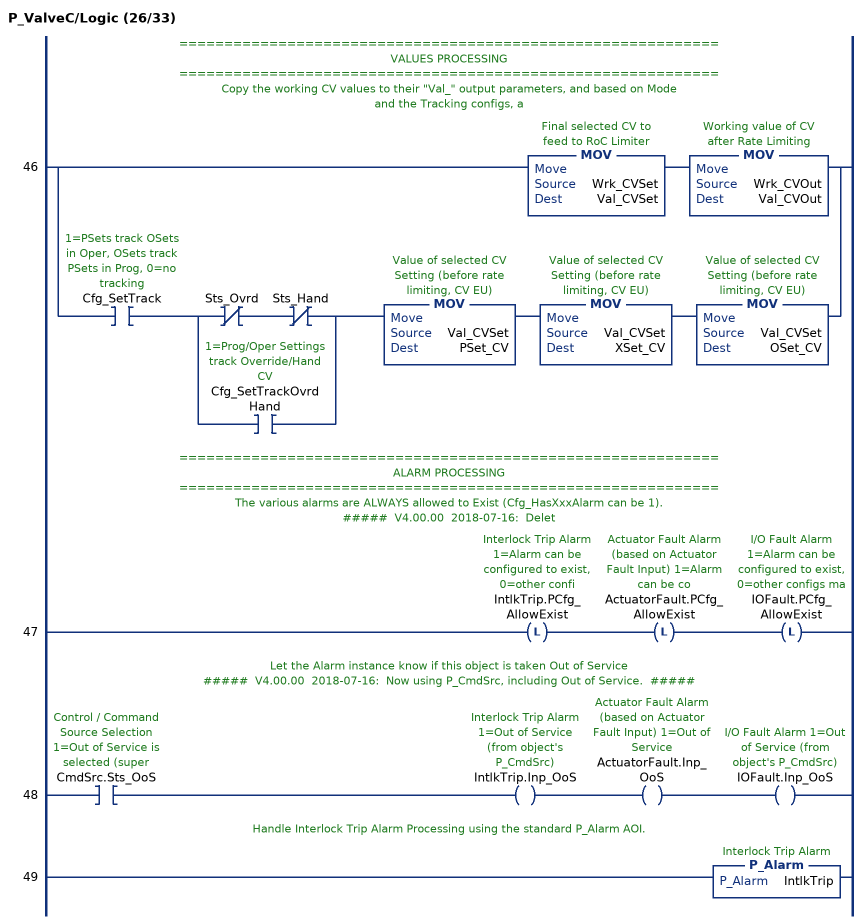
   // ============================================================
   // VALUES PROCESSING
   // ============================================================
   // Copy the working CV values to their "Val_" output parameters, and based on Mode
   // and the Tracking configs, a
   46: [MOV(Wrk_CVSet,Val_CVSet) MOV(Wrk_CVOut,Val_CVOut) ,XIC(Cfg_SetTrack) [XIO(Sts_Ovrd) XIO(Sts_Hand) ,XIC(Cfg_SetTrackOvrdHand) ] MOV(Val_CVSet,PSet_CV) MOV(Val_CVSet,XSet_CV) MOV(Val_CVSet,OSet_CV) ];
   // ============================================================
   // ALARM PROCESSING
   // ============================================================
   // The various alarms are ALWAYS allowed to Exist (Cfg_HasXxxAlarm can be 1).
   // #####  V4.00.00  2018-07-16:  Delet
   47: OTL(IntlkTrip.PCfg_AllowExist)OTL(ActuatorFault.PCfg_AllowExist)OTL(IOFault.PCfg_AllowExist);
   // Let the Alarm instance know if this object is taken Out of Service
   // #####  V4.00.00  2018-07-16:  Now using P_CmdSrc, including Out of Service.  #####
   48: XIC(CmdSrc.Sts_OoS)OTE(IntlkTrip.Inp_OoS)OTE(ActuatorFault.Inp_OoS)OTE(IOFault.Inp_OoS);
   // Handle Interlock Trip Alarm Processing using the standard P_Alarm AOI.
   49: P_Alarm(IntlkTrip);
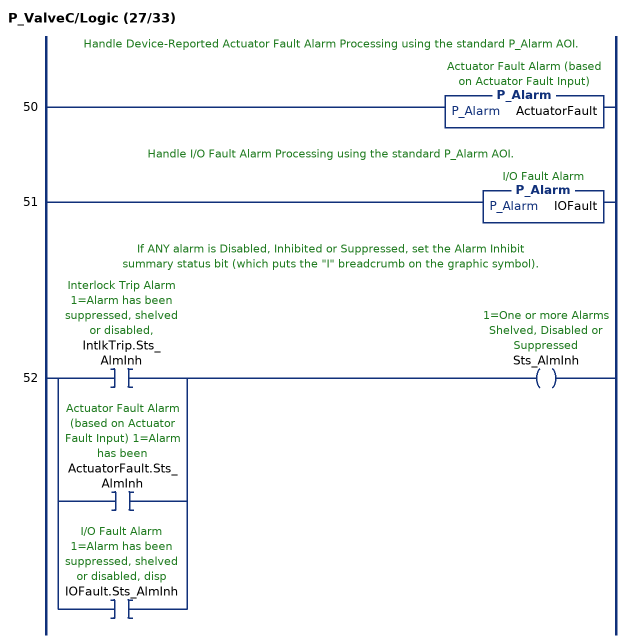
   // Handle Device-Reported Actuator Fault Alarm Processing using the standard P_Alarm AOI.
   50: P_Alarm(ActuatorFault);
   // Handle I/O Fault Alarm Processing using the standard P_Alarm AOI.
   51: P_Alarm(IOFault);
   // If ANY alarm is Disabled, Inhibited or Suppressed, set the Alarm Inhibit
   // summary status bit (which puts the "I" breadcrumb on the graphic symbol).
   52: [XIC(IntlkTrip.Sts_AlmInh) ,XIC(ActuatorFault.Sts_AlmInh) ,XIC(IOFault.Sts_AlmInh) ]OTE(Sts_AlmInh);
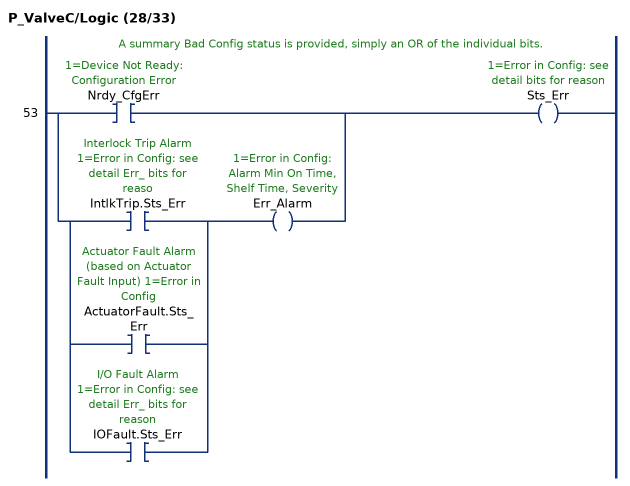
   // A summary Bad Config status is provided, simply an OR of the individual bits.
   53: [XIC(Nrdy_CfgErr) ,[XIC(IntlkTrip.Sts_Err) ,XIC(ActuatorFault.Sts_Err) ,XIC(IOFault.Sts_Err) ] OTE(Err_Alarm) ]OTE(Sts_Err);
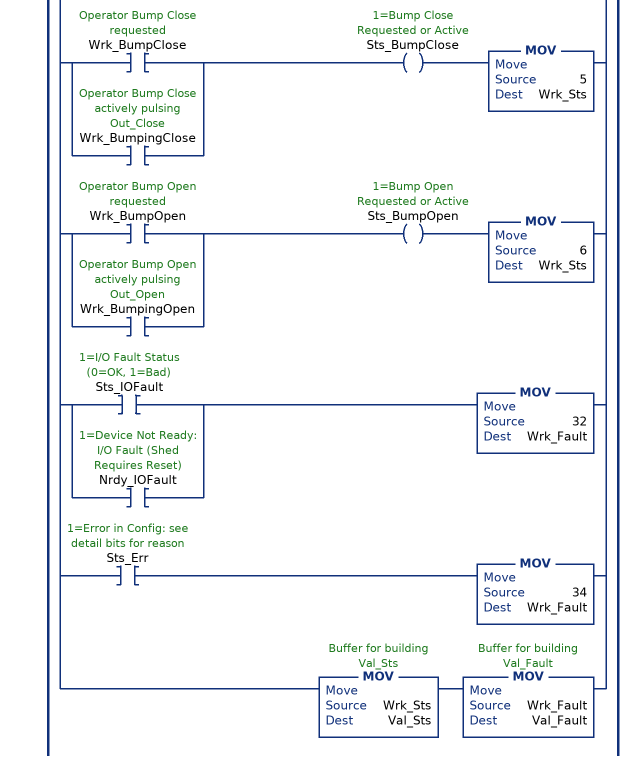
   // This rung generates the enumerated Device Status:
   // 0 = At Target
   // 1 = Ramping Down
   // 2 = Ramping Up
   // 3 = Clamped at CVMin
   // 4 = Clamped at CVMax
   // 5 = Bump Close requested or currently pulsing Out_Close
   // 6 = Bump Open requested or currently pulsing Out_Open
   // And this rung generates the enumerated Device Fault Status:
   // 0 = none
   // 32 = I/O Fault
   // 34 = Configuration Error
   // #####  V4.00.00  2018-07-16:  Disable/Enable replaced by P_CmdSrc Out of Service (OoS).  #####
   54: [CLR(Wrk_Sts) CLR(Wrk_Fault) ,[GRT(Wrk_OpenTime,0.0) XIO(Inp_ActuatorFault) ,XIC(Sts_Ramping) LES(Wrk_CVOut,Wrk_CVSet) ] MOV(2,Wrk_Sts) ,[GRT(Wrk_CloseTime,0.0) XIO(Inp_ActuatorFault) ,XIC(Sts_Ramping) GRT(Wrk_CVOut,Wrk_CVSet) ] MOV(1,Wrk_Sts) ,XIC(Sts_Clamped) [EQU(Wrk_CVOut,Cfg_MinCV) MOV(3,Wrk_Sts) ,EQU(Wrk_CVOut,Cfg_MaxCV) MOV(4,Wrk_Sts) ] ,[XIC(Wrk_BumpClose) ,XIC(Wrk_BumpingClose) ] OTE(Sts_BumpClose) MOV(5,Wrk_Sts) ,[XIC(Wrk_BumpOpen) ,XIC(Wrk_BumpingOpen) ] OTE(Sts_BumpOpen) MOV(6,Wrk_Sts) ,[XIC(Sts_IOFault) ,XIC(Nrdy_IOFault) ] MOV(32,Wrk_Fault) ,XIC(Sts_Err) MOV(34,Wrk_Fault) ,MOV(Wrk_Sts,Val_Sts) MOV(Wrk_Fault,Val_Fault) ];
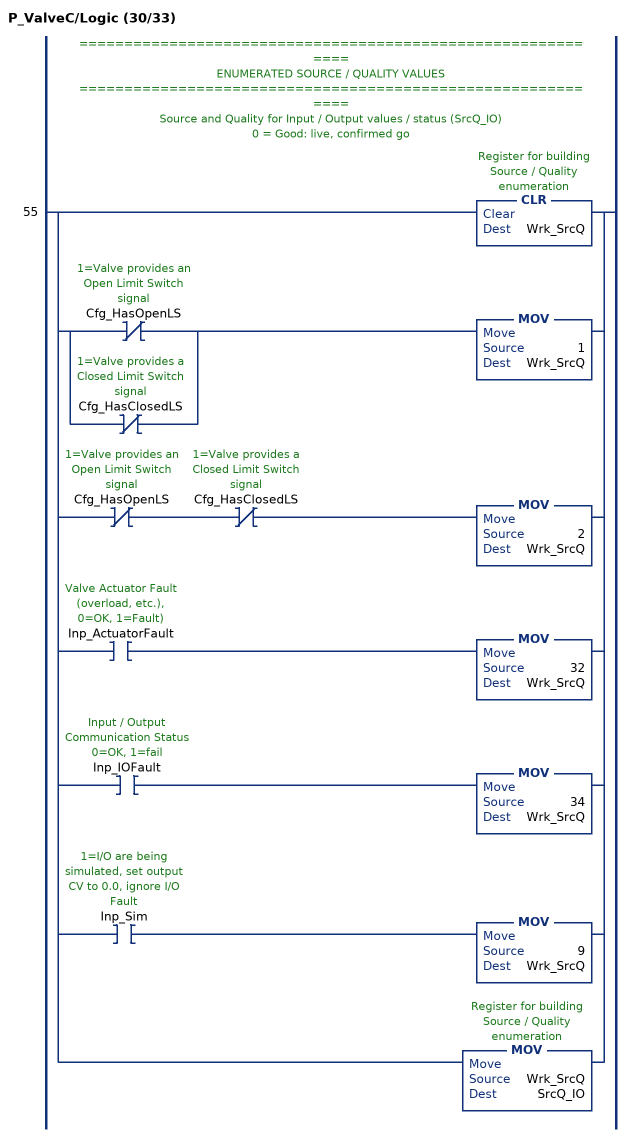
   // ============================================================
   // ENUMERATED SOURCE / QUALITY VALUES
   // ============================================================
   // Source and Quality for Input / Output values / status (SrcQ_IO)
   // 0 = Good: live, confirmed go
   55: [CLR(Wrk_SrcQ) ,[XIO(Cfg_HasOpenLS) ,XIO(Cfg_HasClosedLS) ] MOV(1,Wrk_SrcQ) ,XIO(Cfg_HasOpenLS) XIO(Cfg_HasClosedLS) MOV(2,Wrk_SrcQ) ,XIC(Inp_ActuatorFault) MOV(32,Wrk_SrcQ) ,XIC(Inp_IOFault) MOV(34,Wrk_SrcQ) ,XIC(Inp_Sim) MOV(9,Wrk_SrcQ) ,MOV(Wrk_SrcQ,SrcQ_IO) ];
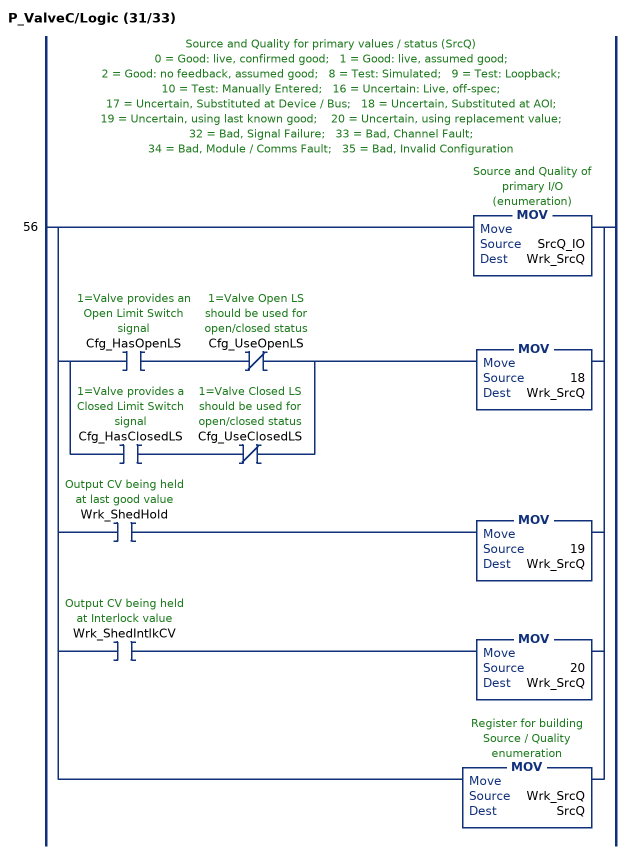
   // Source and Quality for primary values / status (SrcQ)
   // 0 = Good: live, confirmed good;   1 = Good: live, assumed good;
   // 2 = Good: no feedback, assumed good;   8 = Test: Simulated;   9 = Test: Loopback;
   // 10 = Test: Manually Entered;   16 = Uncertain: Live, off-spec;
   // 17 = Uncertain, Substituted at Device / Bus;   18 = Uncertain, Substituted at AOI;
   // 19 = Uncertain, using last known good;    20 = Uncertain, using replacement value;
   // 32 = Bad, Signal Failure;   33 = Bad, Channel Fault;
   // 34 = Bad, Module / Comms Fault;   35 = Bad, Invalid Configuration
   56: [MOV(SrcQ_IO,Wrk_SrcQ) ,[XIC(Cfg_HasOpenLS) XIO(Cfg_UseOpenLS) ,XIC(Cfg_HasClosedLS) XIO(Cfg_UseClosedLS) ] MOV(18,Wrk_SrcQ) ,XIC(Wrk_ShedHold) MOV(19,Wrk_SrcQ) ,XIC(Wrk_ShedIntlkCV) MOV(20,Wrk_SrcQ) ,MOV(Wrk_SrcQ,SrcQ) ];
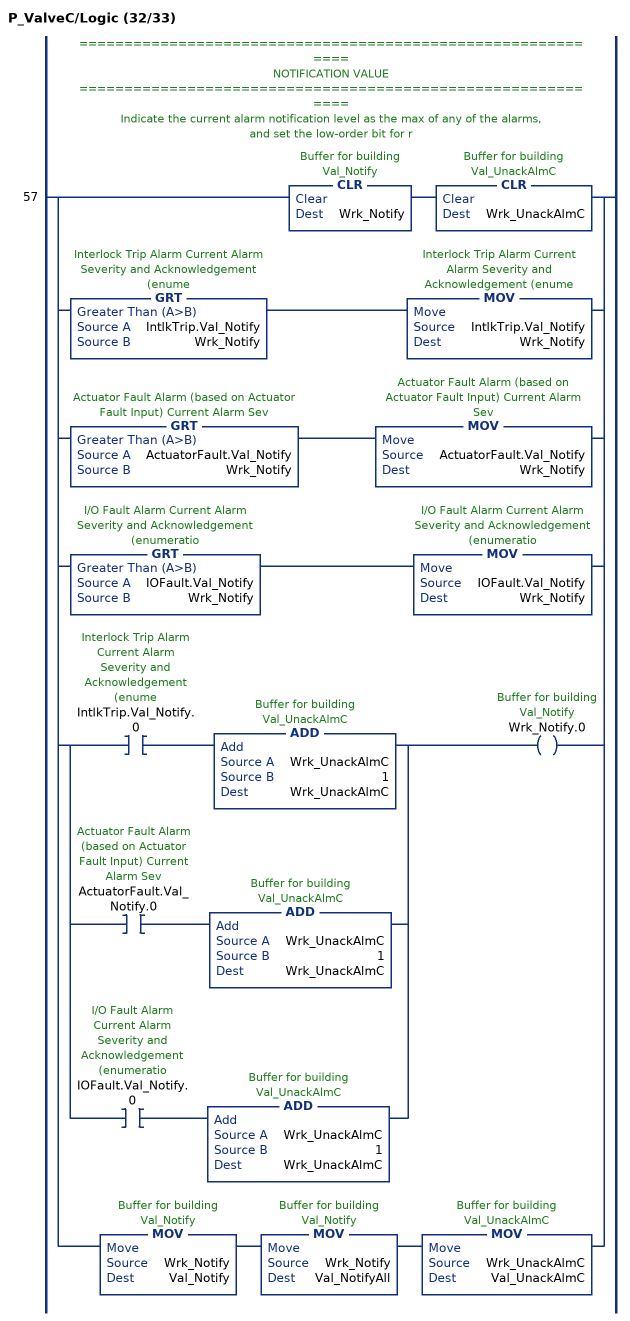
   // ============================================================
   // NOTIFICATION VALUE
   // ============================================================
   // Indicate the current alarm notification level as the max of any of the alarms,
   // and set the low-order bit for r
   57: [CLR(Wrk_Notify) CLR(Wrk_UnackAlmC) ,GRT(IntlkTrip.Val_Notify,Wrk_Notify) MOV(IntlkTrip.Val_Notify,Wrk_Notify) ,GRT(ActuatorFault.Val_Notify,Wrk_Notify) MOV(ActuatorFault.Val_Notify,Wrk_Notify) ,GRT(IOFault.Val_Notify,Wrk_Notify) MOV(IOFault.Val_Notify,Wrk_Notify) ,[XIC(IntlkTrip.Val_Notify.0) ADD(Wrk_UnackAlmC,1,Wrk_UnackAlmC) ,XIC(ActuatorFault.Val_Notify.0) ADD(Wrk_UnackAlmC,1,Wrk_UnackAlmC) ,XIC(IOFault.Val_Notify.0) ADD(Wrk_UnackAlmC,1,Wrk_UnackAlmC) ] OTE(Wrk_Notify.0) ,MOV(Wrk_Notify,Val_Notify) MOV(Wrk_Notify,Val_NotifyAll) MOV(Wrk_UnackAlmC,Val_UnackAlmC) ];
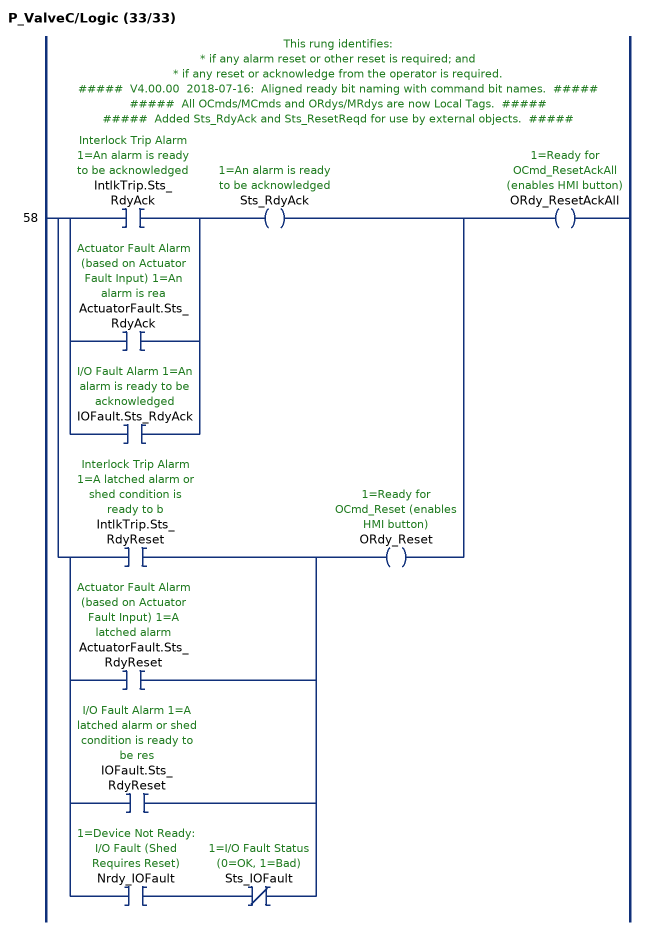
   // This rung identifies:
   // * if any alarm reset or other reset is required; and
   // * if any reset or acknowledge from the operator is required.
   // #####  V4.00.00  2018-07-16:  Aligned ready bit naming with command bit names.  #####
   // #####  All OCmds/MCmds and ORdys/MRdys are now Local Tags.  #####
   // #####  Added Sts_RdyAck and Sts_ResetReqd for use by external objects.  #####
   58: [[XIC(IntlkTrip.Sts_RdyAck) ,XIC(ActuatorFault.Sts_RdyAck) ,XIC(IOFault.Sts_RdyAck) ] OTE(Sts_RdyAck) ,[XIC(IntlkTrip.Sts_RdyReset) ,XIC(ActuatorFault.Sts_RdyReset) ,XIC(IOFault.Sts_RdyReset) ,XIC(Nrdy_IOFault) XIO(Sts_IOFault) ] OTE(ORdy_Reset) ]OTE(ORdy_ResetAckAll);
END_ROUTINE
